FUNCTION Convert_BOOL_TO_TIME : BOOL
VAR_INPUT
	in : BOOL;
	out : REFERENCE TO TIME;
END_VAR
VAR
	converted : TIME;
END_VAR

converted := BOOL_TO_TIME(in);

IF (TIME_TO_BOOL(converted) <> in) THEN
	RETURN;
END_IF

out := converted;
Convert_BOOL_TO_TIME := TRUE;

END_FUNCTION

(* stored: Version 1.1.0.1, ProductVersion 3.1.4024.12
   POU Convert_BOOL_TO_TIME: Id {7d9c4008-6a3f-4a5c-89ad-3aa4f0dc5b34}, SpecialFunc None *)
